(* LS Electric XG5000 project: FLICKER *)
(* PLC LSPLC *)

PROGRAM NewProgram (* task: 스캔 프로그램 *)
VAR
    FLAG : BOOL;
    FLICKER : BOOL;
    FU2 : TOF;
    FUN : TP;
    FUN1 : TON;
    INPUT : BOOL;
    INST : TON;
    INST1 : TOF;
    INST2 : TON_UINT;
    INST3 : TON;
    INST4 : TON;
    INST5 : TOF;
    OFF : TOF;
    OFF1 : TOF;
    OFF2 : TOF;
    ON : TON;
    ON1 : TON;
    ON2 : TON;
    ON3 : TON;
    OUTPUT : BOOL;
    OUTPUT2 : BOOL;
    OUTPUT3 : BOOL;
    PRACTICE1 : BOOL;
    PRACTICE2 : BOOL;
    SOU1 : BOOL;
    SOU2 : BOOL;
    STOP : BOOL;
    SWITCH : BOOL;
    SWITCH2 : BOOL;
    T1 : TON;
    T2 : TON;
    T3 : TON;
    T4 : TON;
    T6 : TON;
    T6_SWITCH : BOOL;
    TIMER1 : TIME;
    TIMER2 : TIME;
    TIMER3 : TIME;
    TIMER4 : TIME;
    TIMER5 : TIME;
    램프5 : BOOL;
    물 : BOOL;
    비데1 : BOOL;
    비데2 : BOOL;
    비데3 : BOOL;
    센서1 : BOOL;
    센서2 : BOOL;
    센서3 : BOOL;
    타이머 : TON;
    타이머1 : TP;
    타이머2 : TP;
    펄스1 : TON;
    펄스2 : TP;
    펄스3 : TOF;
END_VAR

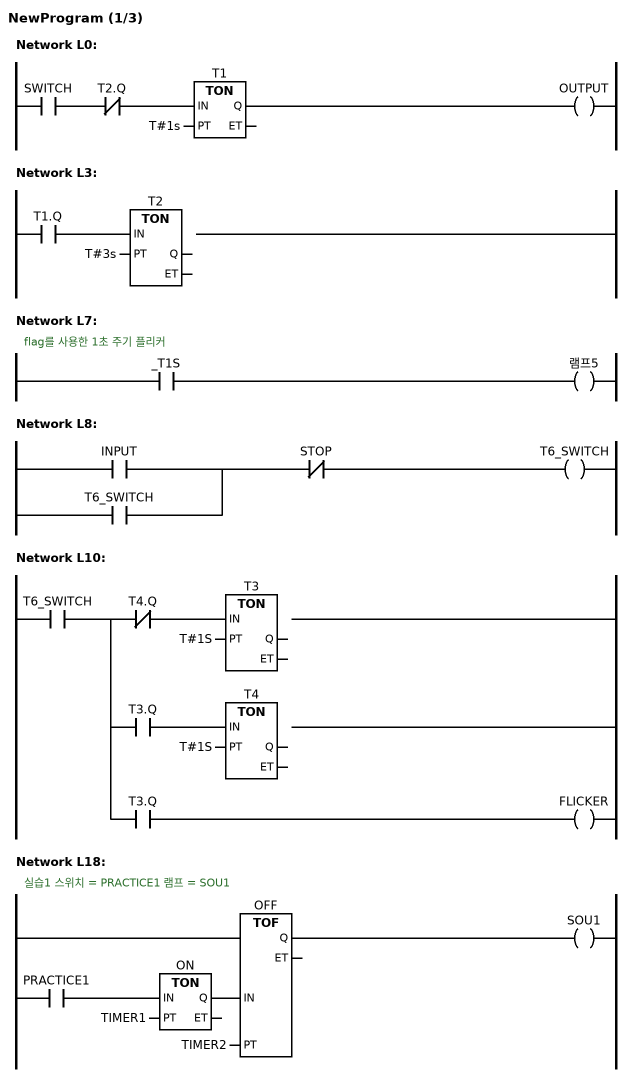
(* Rung L0 *)
T1(IN := SWITCH AND NOT T2.Q, PT := T#1s);
OUTPUT := T1.Q;
(* Rung L3 *)
T2(IN := T1.Q, PT := T#3s);
(* flag를 사용한 1초 주기 플리커 *)
(* Rung L7 *)
램프5 := _T1S;
(* Rung L8 *)
T6_SWITCH := (INPUT OR T6_SWITCH) AND NOT STOP;
(* Rung L10 *)
T3(IN := T6_SWITCH AND NOT T4.Q, PT := T#1S);
T4(IN := T6_SWITCH AND T3.Q, PT := T#1S);
FLICKER := T6_SWITCH AND T3.Q;
(* 실습1 스위치 = PRACTICE1 램프 = SOU1 *)
(* Rung L18 *)
ON(IN := PRACTICE1, PT := TIMER1);
OFF(IN := ON.Q, PT := TIMER2);
SOU1 := OFF.Q;

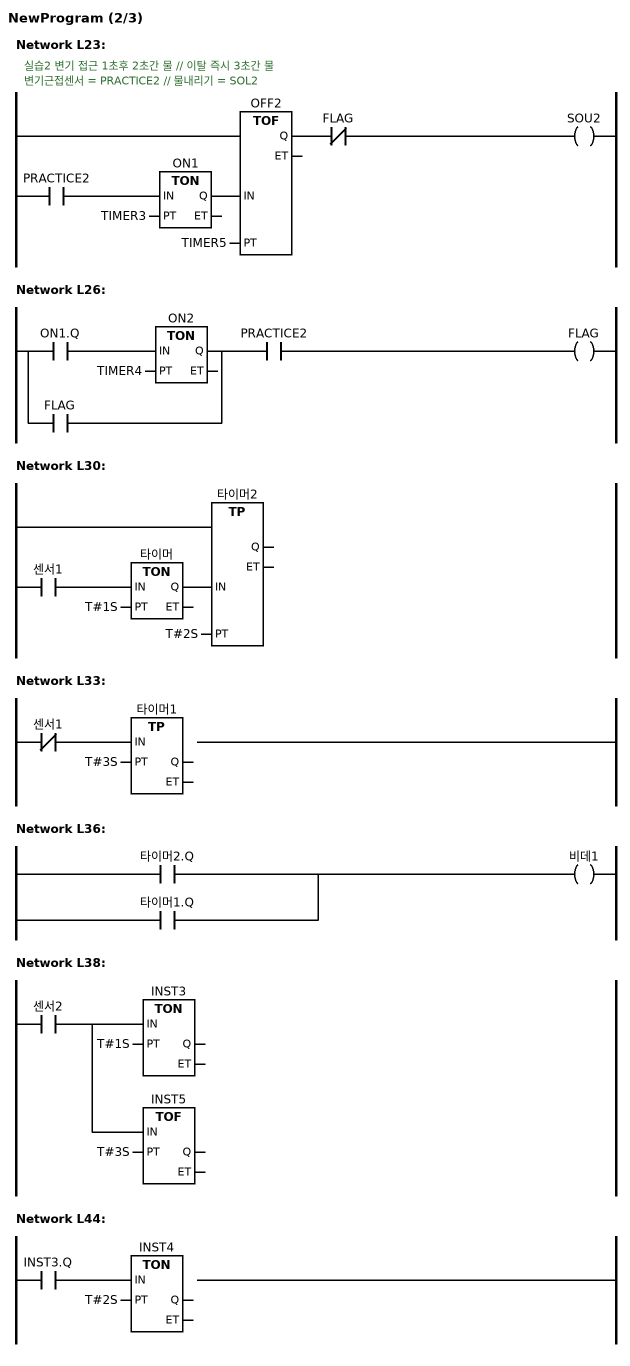
(* 실습2 변기 접근 1초후 2초간 물 // 이탈 즉시 3초간 물 *)
(* 변기근접센서 = PRACTICE2 // 물내리기 = SOL2 *)
(* Rung L23 *)
ON1(IN := PRACTICE2, PT := TIMER3);
OFF2(IN := ON1.Q, PT := TIMER5);
SOU2 := OFF2.Q AND NOT FLAG;
(* Rung L26 *)
ON2(IN := ON1.Q, PT := TIMER4);
FLAG := (ON2.Q OR FLAG) AND PRACTICE2;
(* Rung L30 *)
타이머(IN := 센서1, PT := T#1S);
타이머2(IN := 타이머.Q, PT := T#2S);
(* Rung L33 *)
타이머1(IN := NOT 센서1, PT := T#3S);
(* Rung L36 *)
비데1 := 타이머2.Q OR 타이머1.Q;
(* Rung L38 *)
INST3(IN := 센서2, PT := T#1S);
INST5(IN := 센서2, PT := T#3S);
(* Rung L44 *)
INST4(IN := INST3.Q, PT := T#2S);

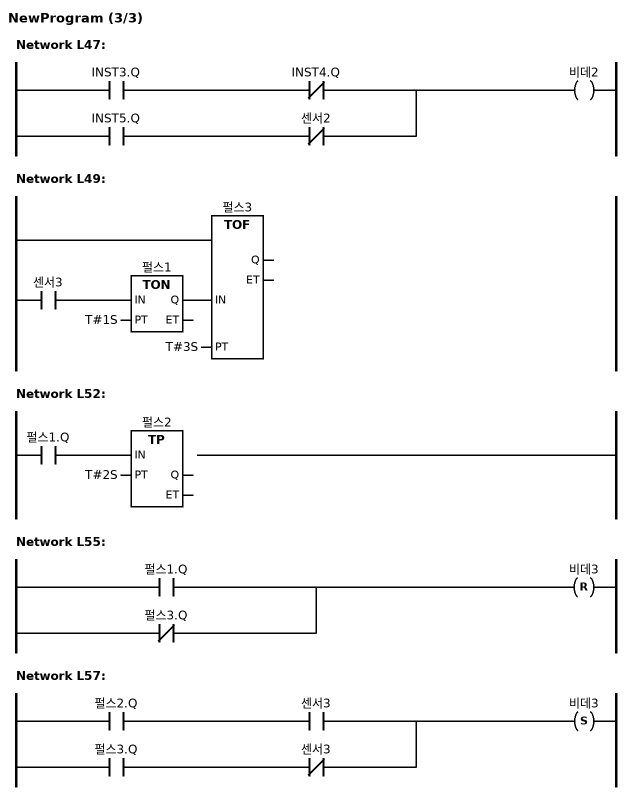
(* Rung L47 *)
비데2 := (INST3.Q AND NOT INST4.Q) OR (INST5.Q AND NOT 센서2);
(* Rung L49 *)
펄스1(IN := 센서3, PT := T#1S);
펄스3(IN := 펄스1.Q, PT := T#3S);
(* Rung L52 *)
펄스2(IN := 펄스1.Q, PT := T#2S);
(* Rung L55 *)
IF 펄스1.Q OR NOT 펄스3.Q THEN 비데3 := FALSE; END_IF;
(* Rung L57 *)
IF (펄스2.Q AND 센서3) OR (펄스3.Q AND NOT 센서3) THEN 비데3 := TRUE; END_IF;
END_PROGRAM